{attribute addProperty BoxType "EL2212-0000-0018"}
{attribute addProperty Id "ControlAT %Q*Control_4A122216162"}
{attribute addProperty CRC "206303623"}
{attribute addProperty SizeInBites "16"}
{attribute addProperty SizeInBytes "2"}
TYPE DOX_Control_Channel_0C4BF187 :
STRUCT
	{attribute addProperty Name "Control"}
	Control AT %Q* : Control_4A122216;
END_STRUCT
END_TYPE

(* stored: Version 1.2.0.0, ProductVersion 3.1.4024.9
   DUT DOX_Control_Channel_0C4BF187: Id {f1cfdb70-7fea-4be0-9d21-f4b3a5274aeb} *)
